FUNCTION_BLOCK FB_Idle IMPLEMENTS I_State
VAR_INPUT
END_VAR
VAR_OUTPUT
END_VAR
VAR
	pAxis : POINTER TO FB_Axis;
END_VAR

{warning 'add method implementation '}
METHOD Disable : BOOL
END_METHOD

{warning 'add method implementation '}
METHOD Enable : BOOL
END_METHOD

METHOD FB_init : BOOL
VAR_INPUT
	bInitRetains : BOOL; // if TRUE, the retain variables are initialized (warm start / cold start)
	bInCopyCode : BOOL;  // if TRUE, the instance afterwards gets moved into the copy code (online change)
	pAxis : POINTER TO FB_Axis;
END_VAR
THIS^.pAxis := pAxis;
END_METHOD

{warning 'add method implementation '}
METHOD Reset : BOOL
END_METHOD

END_FUNCTION_BLOCK

(* stored: Version 1.1.0.1, ProductVersion 3.1.4024.3
   POU FB_Idle: Id {e98a13b5-3373-4c7e-b54b-aedb08bbf98f}, SpecialFunc None
   Method Disable: Id {a3c10d82-0675-42d9-98a3-2caa21feda67}
   Method Enable: Id {3efa1120-c0a5-4ccb-9e2b-52976746f615}
   Method FB_init: Id {606ceec6-c0ac-43a1-94cb-6490b257ef3c}
   Method Reset: Id {6f1d9d75-58e1-4a5f-adcd-6f685e14c158} *)
